TYPE ST_EquipmentModuleFaults :
STRUCT
	ipEquipmentFault1 : I_Fault;
END_STRUCT
END_TYPE

(* stored: Version 1.1.0.1, ProductVersion 3.1.4026.18
   DUT ST_EquipmentModuleFaults: Id {b9c2cdf4-6702-45d3-804b-a1ef1760174c} *)
